// TIA Portal V20 export
FUNCTION "CallEnergy" : Void   // FC5, LAD
TITLE = CallEnergy
// Call of Demo EnergyMeter and Energy Efficient M for EEMM demonstration
// stored: IsIECCheckEnabled true, SetENOAutomatically true
BEGIN

REGION Network 1: BLOCK INFO HEADER
   // SIEMENS AG / (c)Copyright 2023
   // ------------------------------------------------------------------------------
   // Title:            CallEnergy (FC5)
   // Comment/Function: Call of Demo EnergyMeter and Energy Efficient M for EEMM demonstration
   // Library/Family:   Energy
   // Author:           SICAR
   // Tested with:      ---
   // Engineering:      TIA Portal V19
   // Restrictions:     -
   // Requirements:     ---
   // ------------------------------------------------------------------------------
   // Change log table:
   // Version  | Date       | Expert in charge       | Changes applied
   // ---------|------------|------------------------|------------------------------
   // 01.00.00 | 11.12.2023 | SICAR
   //                         First released version
END_REGION

REGION Network 2: Call: Demo EnergyMeter, Energy Efficient M
   // Call for EEM demonstration
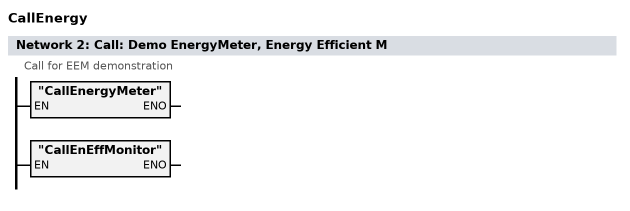
   RUNG wire#powerrail
      "CallEnergyMeter"()
   END_RUNG
   RUNG wire#powerrail
      "CallEnEffMonitor"()
   END_RUNG
   // the same network as SCL:
   "CallEnergyMeter"();
   "CallEnEffMonitor"();
END_REGION

REGION Network 3: Empty
END_REGION
END_FUNCTION
